// TwinCAT 3 PLC project PRG_B_Base_HMI
// Title: B_Base_HMI_Connector
// Company: RafalOS
// Author: Rafał Osajda
// ProjectVersion: 0.0.1.00
// ProgramVersion: 3.1.4026.18
// libraries:
//   B_Base, * (RafalOS)
//   Tc2_Standard, * (Beckhoff Automation GmbH)
//   Tc2_System, * (Beckhoff Automation GmbH)
//   Tc3_Module, * (Beckhoff Automation GmbH)
// project tree:
//   DUTs/ ST_BaseHMIDescriptor.TcDUT, ST_BaseHMIDescriptorEdit.TcDUT, ST_ListOfElement_HMI.TcDUT, ST_RowListOfElement_HMI.TcDUT
//   / PlcTask.TcTTO (not stored)
//   POUs Compilation/ PRG_Compilation.TcPOU
//   POUs/A02_FB_BaseHMILogger/ FB_BaseHMILogger.TcPOU, ITF_BaseHMILogger.TcIO, ST_BaseHMILogger.TcDUT
//   POUs/A03a_FB_BaseHMILoggerElement_View/ FB_BaseHMILoggerElement_View.TcPOU, ITF_BaseHMILoggerElement_View.TcIO, ST_BaseHMIConnectorEvents_ActionButtuns.TcDUT (not stored), ST_BaseHMIConnectorEvents_DetailInformation.TcDUT (not stored), ST_BaseHMIConnectorEvents_Filter.TcDUT (not stored), ST_BaseHMIConnectorEvents_ListToDisplay.TcDUT, ST_BaseHMILoggerElement_View.TcDUT, ST_BaseHMIConnectorEvents_ListToDisplayRow.TcDUT (not stored)
//   POUs/A03b_FB_BaseHMILoggerElement_Command/ FB_BaseHMILoggerElement_Command.TcPOU, ITF_BaseHMILoggerElement_Command.TcIO, ST_BaseHMILoggerElement_Command_DataCheck.TcDUT, ST_BaseHMILoggerElement_Command.TcDUT
//   POUs/A04a_FB_BaseHMIComponent_View/ FB_BaseHMIComponent_View.TcPOU, ITF_BaseHMIComponent_View.TcIO, ST_BaseHMIComponent_View.TcDUT, ST_BaseHMIComponent_View_Link.TcDUT
//   POUs/A04b_FB_BaseHMIComponent_Command/ FB_BaseHMIComponent_Command.TcPOU, ITF_BaseHMIComponent_Command.TcIO, ST_BaseHMIComponent_Command.TcDUT, ST_BaseHMIComponent_Command_Link.TcDUT
//   POUs/A05a_FB_BaseHMIControlElement_View/ FB_BaseHMIControlElement_View.TcPOU, ITF_BaseHMIControlElement_View.TcIO, ST_BaseHMIControlElement_View.TcDUT, ST_BaseHMIControlElement_View_Link.TcDUT
//   POUs/A05b_FB_BaseHMIControlElement_Command/ FB_BaseHMIControlElement_Command.TcPOU, ITF_BaseHMIControlElement_Command.TcIO, ST_BaseHMIControlElement_Command.TcDUT, ST_BaseHMIControlElement_Command_Link.TcDUT
//   POUs/A06a_FB_BaseHMIGroupElement_View/ FB_BaseHMIGroupElement_View.TcPOU, ITF_BaseHMIGroupElement_View.TcIO, ST_BaseHMIGroupElement_View.TcDUT, ST_BaseHMIGroupElement_View_Link.TcDUT
//   POUs/A06b_FB_BaseHMIGroupElement_Command/ FB_BaseHMIGroupElement_Command.TcPOU, ITF_BaseHMIGroupElement_Command.TcIO, ST_BaseHMIGroupElement_Command.TcDUT, ST_BaseHMIGroupElement_Command_Link.TcDUT
//   POUs/A07a_FB_BaseHMITopElement_View/ FB_BaseHMITopElement_View.TcPOU, ITF_BaseHMITopElement_View.TcIO, ST_BaseHMITopElement_View.TcDUT, ST_BaseHMITopElement_View_Link.TcDUT
//   POUs/A07b_FB_BaseHMITopElement_Command/ FB_BaseHMITopElement_Command.TcPOU, ITF_BaseHMITopElement_Command.TcIO, ST_BaseHMITopElement_Command.TcDUT, ST_BaseHMITopElement_Command_Link.TcDUT
//   POUs/B02_Recipe/ FB_BaseRecipe_HMI.TcPOU, ITF_BaseRecipe_HMI.TcIO, ST_BaseRecipe_HMI.TcDUT
// real-time tasks:
//   TASK PlcTask: cycle T#10ms, priority 20, ADS port 350

// ---- DUTs/ST_BaseHMIDescriptor.TcDUT
TYPE ST_BaseHMIDescriptor :
STRUCT
	wsText						: WSTRING;
	sUnit						: STRING(6);
	rValue						: REAL;
	rMin						: REAL;
	rMax						: REAL;
	rDefaultValue				: REAL;
END_STRUCT
END_TYPE

// ---- DUTs/ST_BaseHMIDescriptorEdit.TcDUT
TYPE ST_BaseHMIDescriptorEdit :
STRUCT
	wsText						: WSTRING;
	sUnit						: STRING(6);
	rValue						: REAL;
	rMin						: REAL;
	rMax						: REAL;
	rDefaultValue				: REAL;
	rValueOld					: REAL; //wartosc przed zmiana do porównania czy cos się zmieniło
	bSave						: BOOL;
	bSetDefault					: BOOL;
	bCancel						: BOOL;
	bVisibleSave				: BOOL;
	bVisibleSetDefault			: BOOL;
	bVisibleCancel				: BOOL;
	iID							: int; //numer deskryptora do edycji
END_STRUCT
END_TYPE

// ---- DUTs/ST_ListOfElement_HMI.TcDUT
TYPE ST_ListOfElement_HMI :
STRUCT
(*	Lista wszystkich dodanych komponentów 	*)
	arrRow					: ARRAY [1..GVL_BaseConstans.MAX_NUMBER_OF_ALL_ITEM] OF ST_RowListOfElement_HMI;
	iNumberOfAdded			: INT;
(*	Lista indeksów PB w tablicy arrWiersz	*)
	arrRowOfListTE			: ARRAY [1..GVL_BaseConstans.MAX_NUMBER_OF_TOP_ELEMENT] OF INT;
	iNumberOfAddedTE		: INT;
END_STRUCT
END_TYPE

// ---- DUTs/ST_RowListOfElement_HMI.TcDUT
TYPE ST_RowListOfElement_HMI :
STRUCT
	stIdentifiers		: ST_BaseElementIdentifier;
	itfElement			: ITF_BaseHMIComponent_View;
//
	arrChild			: ARRAY [0..GVL_BaseConstans.MAX_ITEM_PER_ELEMENT] OF INT;
	iNumberOfChildAdded	: INT;
	
END_STRUCT
END_TYPE

// ---- POUs/A02_FB_BaseHMILogger/ST_BaseHMILogger.TcDUT
TYPE ST_BaseHMILogger :
STRUCT
	bDanaBaseLogger		: BOOL;
END_STRUCT
END_TYPE

// ---- POUs/A03a_FB_BaseHMILoggerElement_View/ST_BaseHMIConnectorEvents_ListToDisplay.TcDUT
TYPE ST_BaseHMIConnectorEvents_ListToDisplay :
STRUCT
	arrToDisplay				: ARRAY [1..GVL_BaseConstans.MAX_EVENTS_TO_SHOW] OF ST_BaseHMIConnectorEvents_ListToDisplayRow;
	iNumberOfRow				: INT;

END_STRUCT
END_TYPE

// ---- POUs/A03a_FB_BaseHMILoggerElement_View/ST_BaseHMILoggerElement_View.TcDUT
TYPE ST_BaseHMILoggerElement_View :
STRUCT
	stFilter						: ST_BaseHMIConnectorEvents_Filter;
	stListOfEventsToDisplay			: ST_BaseHMIConnectorEvents_ListToDisplay;
	stButtons						: ST_BaseHMIConnectorEvents_ActionButtuns;
	stDetailInformation				: ST_BaseHMIConnectorEvents_DetailInformation;
	bSelected						: BOOL;
	iSelectedRow					: INT;
	iSelectedRowPrevius				: INT;
	bRefreshInfo					: BOOL;
	bRefreshList					: BOOL;
	
END_STRUCT
END_TYPE

// ---- POUs/A03b_FB_BaseHMILoggerElement_Command/ST_BaseHMILoggerElement_Command_DataCheck.TcDUT
TYPE ST_BaseHMILoggerElement_Command_DataCheck :
STRUCT
	eMode			: REFERENCE TO E_BaseMachineMode;	//tryb pracy
	bSafety			: REFERENCE TO BOOL;	//ogólna flaga czy safety pozwala na pracę 
END_STRUCT
END_TYPE

// ---- POUs/A03b_FB_BaseHMILoggerElement_Command/ST_BaseHMILoggerElement_Command.TcDUT
TYPE ST_BaseHMILoggerElement_Command :
STRUCT
END_STRUCT
END_TYPE

// ---- POUs/A04a_FB_BaseHMIComponent_View/ST_BaseHMIComponent_View.TcDUT
TYPE ST_BaseHMIComponent_View :
STRUCT
	wsName			: WSTRING;
	
END_STRUCT
END_TYPE

// ---- POUs/A04a_FB_BaseHMIComponent_View/ST_BaseHMIComponent_View_Link.TcDUT
(*			
	RAFALOS
	Rafał Osajda		23.09.2025		TC 4024.66
	Struktura pomocnicza potrzeba do wiazania zmiennych
*)
TYPE ST_BaseHMIComponent_View_Link :
STRUCT
	stLoggerElement				: ST_BaseHMILoggerElement_View;
	stComponent					: ST_BaseHMIComponent_View;
END_STRUCT
END_TYPE

// ---- POUs/A04b_FB_BaseHMIComponent_Command/ST_BaseHMIComponent_Command.TcDUT
TYPE ST_BaseHMIComponent_Command :
STRUCT
END_STRUCT
END_TYPE

// ---- POUs/A04b_FB_BaseHMIComponent_Command/ST_BaseHMIComponent_Command_Link.TcDUT
(*			
	RAFALOS
	Rafał Osajda		23.09.2025		TC 4024.66
	Struktura pomocnicza potrzeba do wiazania zmiennych
*)
TYPE ST_BaseHMIComponent_Command_Link :
STRUCT
	stLoggerElement				: ST_BaseHMILoggerElement_Command;
	stComponent					: ST_BaseHMIComponent_Command;
END_STRUCT
END_TYPE

// ---- POUs/A05a_FB_BaseHMIControlElement_View/ST_BaseHMIControlElement_View.TcDUT
TYPE ST_BaseHMIControlElement_View :
STRUCT
	bDanaBaseControlElement		: BOOL;
	
END_STRUCT
END_TYPE

// ---- POUs/A05a_FB_BaseHMIControlElement_View/ST_BaseHMIControlElement_View_Link.TcDUT
(*			
	RAFALOS
	Rafał Osajda		23.09.2025		TC 4024.66
	Struktura pomocnicza potrzeba do wiazania zmiennych
*)
TYPE ST_BaseHMIControlElement_View_Link :
STRUCT
	stLoggerElement				: ST_BaseHMILoggerElement_View;
	stComponent					: ST_BaseHMIComponent_View;
	stControlElement			: ST_BaseHMIControlElement_View;
END_STRUCT
END_TYPE

// ---- POUs/A05b_FB_BaseHMIControlElement_Command/ST_BaseHMIControlElement_Command.TcDUT
TYPE ST_BaseHMIControlElement_Command :
STRUCT
END_STRUCT
END_TYPE

// ---- POUs/A05b_FB_BaseHMIControlElement_Command/ST_BaseHMIControlElement_Command_Link.TcDUT
TYPE ST_BaseHMIControlElement_Command_Link :
STRUCT
	stLoggerElement				: ST_BaseHMILoggerElement_Command;
	stComponent					: ST_BaseHMIComponent_Command;
	stControlElement			: ST_BaseHMIControlElement_Command;
END_STRUCT
END_TYPE

// ---- POUs/A06a_FB_BaseHMIGroupElement_View/ST_BaseHMIGroupElement_View.TcDUT
TYPE ST_BaseHMIGroupElement_View :
STRUCT
	bDanaBaseGroupElement		: BOOL;
END_STRUCT
END_TYPE

// ---- POUs/A06a_FB_BaseHMIGroupElement_View/ST_BaseHMIGroupElement_View_Link.TcDUT
(*			
	RAFALOS
	Rafał Osajda		23.09.2025		TC 4024.66
	Struktura pomocnicza potrzeba do wiazania zmiennych
*)
TYPE ST_BaseHMIGroupElement_View_Link :
STRUCT
	stLoggerElement				: ST_BaseHMILoggerElement_View;
	stComponent					: ST_BaseHMIComponent_View;
	stControlElement			: ST_BaseHMIControlElement_View;
	stGroupElement				: ST_BaseHMIGroupElement_View;
END_STRUCT
END_TYPE

// ---- POUs/A06b_FB_BaseHMIGroupElement_Command/ST_BaseHMIGroupElement_Command.TcDUT
TYPE ST_BaseHMIGroupElement_Command :
STRUCT
END_STRUCT
END_TYPE

// ---- POUs/A06b_FB_BaseHMIGroupElement_Command/ST_BaseHMIGroupElement_Command_Link.TcDUT
TYPE ST_BaseHMIGroupElement_Command_Link :
STRUCT
	stLoggerElement				: ST_BaseHMILoggerElement_Command;
	stComponent					: ST_BaseHMIComponent_Command;
	stControlElement			: ST_BaseHMIControlElement_Command;
	stGroupElement				: ST_BaseHMIGroupElement_Command;
END_STRUCT
END_TYPE

// ---- POUs/A07a_FB_BaseHMITopElement_View/ST_BaseHMITopElement_View.TcDUT
TYPE ST_BaseHMITopElement_View :
STRUCT
	bDanaTopElement				: BOOL;
END_STRUCT
END_TYPE

// ---- POUs/A07a_FB_BaseHMITopElement_View/ST_BaseHMITopElement_View_Link.TcDUT
(*			
	RAFALOS
	Rafał Osajda		23.09.2025		TC 4024.66
	Struktura pomocnicza potrzeba do wiazania zmiennych
*)
TYPE ST_BaseHMITopElement_View_Link :
STRUCT
	stLoggerElement				: ST_BaseHMILoggerElement_View;
	stComponent					: ST_BaseHMIComponent_View;
	stControlElement			: ST_BaseHMIControlElement_View;
	stGroupElement				: ST_BaseHMIGroupElement_View;
	stTopElement				: ST_BaseHMITopElement_View;
END_STRUCT
END_TYPE

// ---- POUs/A07b_FB_BaseHMITopElement_Command/ST_BaseHMITopElement_Command.TcDUT
TYPE ST_BaseHMITopElement_Command :
STRUCT
END_STRUCT
END_TYPE

// ---- POUs/A07b_FB_BaseHMITopElement_Command/ST_BaseHMITopElement_Command_Link.TcDUT
TYPE ST_BaseHMITopElement_Command_Link :
STRUCT
	stLoggerElement				: ST_BaseHMILoggerElement_Command;
	stComponent					: ST_BaseHMIComponent_Command;
	stControlElement				: ST_BaseHMIControlElement_Command;
	stGroupElement				: ST_BaseHMIGroupElement_Command;
	stTopElement					: ST_BaseHMITopElement_Command;
END_STRUCT
END_TYPE

// ---- POUs/B02_Recipe/ST_BaseRecipe_HMI.TcDUT
TYPE ST_BaseRecipe_HMI :
STRUCT
END_STRUCT
END_TYPE

// ---- POUs/A02_FB_BaseHMILogger/ITF_BaseHMILogger.TcIO
INTERFACE ITF_BaseHMILogger

END_INTERFACE

// ---- POUs/A03a_FB_BaseHMILoggerElement_View/ITF_BaseHMILoggerElement_View.TcIO
INTERFACE ITF_BaseHMILoggerElement_View

(*			
	RafalOS
	Rafał Osajda		19.11.2025		TC 4024.66
	Czyści danych przy zmienia ramki po poprzedniej ramce
*)
METHOD PUBLIC ClearAfterScreen : BOOL
VAR_INPUT
END_VAR
END_METHOD

(*			
	EVERDE sp. z o.o.
	Rafał Osajda		09.09.2025		TC 4024.66
	Generuje tablicę zdarzeń dla podanego ID dla 0 dla wszystkich elementów
*)
METHOD PUBLIC GetEventTableForIDItem : BOOL
VAR_INPUT
	uiIdItem			: UINT;
END_VAR
END_METHOD

(*			
	EVERDE sp. z o.o.
	Rafał Osajda		09.09.2025		TC 4024.66
	Zwraca tablicę swoich zdarzeń
*)
METHOD PUBLIC GetYourEventTable : BOOL
VAR_INPUT
END_VAR
END_METHOD

(*			
	RafalOS
	Rafał Osajda		14.11.2025		TC 4024.66
	Metoda przygotowywania danych dla HMI 
	W niej odbywa się odpytywanie właściego elementu przez łącznik
*)
METHOD PUBLIC PrepareDataForHMI : BOOL
VAR_INPUT
END_VAR
END_METHOD

(*			
	RafalOS
	Rafał Osajda		19.11.2025		TC 4024.66
	Przygotowanie ramki pood tamke do wyświetlenia - tylko przygotowanie a nie przygotowanie danych do wyświetlenia
*)
METHOD PUBLIC PrepareForScreen : BOOL
VAR_INPUT
END_VAR
END_METHOD

END_INTERFACE

// ---- POUs/A03b_FB_BaseHMILoggerElement_Command/ITF_BaseHMILoggerElement_Command.TcIO
INTERFACE ITF_BaseHMILoggerElement_Command

END_INTERFACE

// ---- POUs/A04a_FB_BaseHMIComponent_View/ITF_BaseHMIComponent_View.TcIO
INTERFACE ITF_BaseHMIComponent_View EXTENDS ITF_BaseHMILoggerElement_View

METHOD PUBLIC IsValidCommonData : BOOL
VAR_INPUT
END_VAR
END_METHOD

METHOD PUBLIC JoinTheList : INT
VAR_INPUT
	refstList				: REFERENCE TO ST_ListOfElement_HMI;
	iNumberOfParent			: INT; 	//numer rodzica na liście
END_VAR
END_METHOD

METHOD PUBLIC LinkCommonData : BOOL
VAR_INPUT
	stCommonData				: REFERENCE TO ST_BaseCommonData;
END_VAR
END_METHOD

END_INTERFACE

// ---- POUs/A04b_FB_BaseHMIComponent_Command/ITF_BaseHMIComponent_Command.TcIO
INTERFACE ITF_BaseHMIComponent_Command EXTENDS ITF_BaseHMILoggerElement_Command

END_INTERFACE

// ---- POUs/A05a_FB_BaseHMIControlElement_View/ITF_BaseHMIControlElement_View.TcIO
INTERFACE ITF_BaseHMIControlElement_View EXTENDS ITF_BaseHMIComponent_View

END_INTERFACE

// ---- POUs/A05b_FB_BaseHMIControlElement_Command/ITF_BaseHMIControlElement_Command.TcIO
INTERFACE ITF_BaseHMIControlElement_Command EXTENDS ITF_BaseHMIComponent_Command

END_INTERFACE

// ---- POUs/A06a_FB_BaseHMIGroupElement_View/ITF_BaseHMIGroupElement_View.TcIO
INTERFACE ITF_BaseHMIGroupElement_View EXTENDS ITF_BaseHMIControlElement_View

END_INTERFACE

// ---- POUs/A06b_FB_BaseHMIGroupElement_Command/ITF_BaseHMIGroupElement_Command.TcIO
INTERFACE ITF_BaseHMIGroupElement_Command EXTENDS ITF_BaseHMIControlElement_Command

END_INTERFACE

// ---- POUs/A07a_FB_BaseHMITopElement_View/ITF_BaseHMITopElement_View.TcIO
INTERFACE ITF_BaseHMITopElement_View EXTENDS ITF_BaseHMIComponent_View

END_INTERFACE

// ---- POUs/A07b_FB_BaseHMITopElement_Command/ITF_BaseHMITopElement_Command.TcIO
INTERFACE ITF_BaseHMITopElement_Command EXTENDS ITF_BaseHMIGroupElement_Command

END_INTERFACE

// ---- POUs/B02_Recipe/ITF_BaseRecipe_HMI.TcIO
INTERFACE ITF_BaseRecipe_HMI EXTENDS ITF_Base

(*			
	RafalOS
	Rafał Osajda		03.03.2025		TC 4026.13		wer. 0.0.0.1
	Kopiuje składniki z wybranej receptury i tworzy nową recepture
*)
METHOD PUBLIC AddRecipeFromRecipe : BOOL
VAR_INPUT
	uiNumberRecipe				: UINT;
	stTexts						: ST_BaseLabel;
END_VAR
END_METHOD

(*			
	RafalOS
	Rafał Osajda		03.03.2025		TC 4026.13		wer. 0.0.0.1
	Kopiuje składniki z wybranego szablonu i tworzy nową recepture
*)
METHOD PUBLIC AddRecipeFromTemplate : BOOL
VAR_INPUT
	uiNumberTemplates			: UINT;
	stTexts						: ST_BaseLabel;
END_VAR
END_METHOD

(*			
	RafalOS
	Rafał Osajda		03.06.2025		TC 4024.66
	usuwa referencje do wybranej
*)
METHOD PUBLIC ClearChosen
VAR_INPUT
END_VAR
END_METHOD

(*			
	RafalOS
	Rafał Osajda		25.10.2025		TC 4024.66
	Utworzenie nowych szablonów receptur na podstawie dodanych fb zewnętrznych - wywołanie metody powoduje
	skosowanie dotychczasowych szablonów i receptur
*)
METHOD PUBLIC CreateRecipeTemplates : BOOL
VAR_INPUT
END_VAR
END_METHOD

(*			
	RafalOS
	Rafał Osajda		03.03.2025		TC 4026.13		wer. 0.0.0.1
	
*)
METHOD PUBLIC DeleteRecipe : BOOL
VAR_INPUT
	uiNumber				: uint;
END_VAR
END_METHOD

(*			
	RafalOS
	Rafał Osajda		03.03.2025		TC 4026.13		wer. 0.0.0.1
	
*)
METHOD PUBLIC GetIngredientFromRecipe : ST_BaseDescriptor
VAR_INPUT
	uiNumberOfRecipe			: UINT;
	uiNumberOfIngredient		: UINT;
END_VAR
END_METHOD

(*			
	RafalOS
	Rafał Osajda		02.12.2025		TC 4024.66
	Zwraca do tablicy wybrany zakres składników
*)
METHOD PUBLIC GetIngredientRange 
VAR_INPUT
	iRecipe			: INT;	//numer receptury z której bierzemy składniki
	iStartIndex		: INT;	//numer startowy składnika
	iCount			: INT;	//ilośc pobieranych 
END_VAR
VAR_IN_OUT
	arrOut : ARRAY [*] OF ST_BaseDescriptor;
END_VAR
VAR_OUTPUT
	iNumberOfFilledData	: INT;	//ilosc wypelnionych danych na strone
END_VAR
END_METHOD

METHOD GetNameList : ST_BaseRecipeList
VAR_INPUT
END_VAR
END_METHOD

METHOD GetNameListTemplate : ST_BaseRecipeList
VAR_INPUT
END_VAR
END_METHOD

METHOD GetNamesOfSelectRecipe : ST_BaseLabel
VAR_INPUT

END_VAR
END_METHOD

(*			
	RafalOS
	Rafał Osajda		03.03.2025		TC 4026.13		wer. 0.0.0.1
	
*)
METHOD PUBLIC GetNumberIngredientOfRecipe : UINT
VAR_INPUT
	uiNumber				: UINT;
END_VAR
END_METHOD

METHOD PUBLIC GetNumberOfChoosen : UINT
VAR_INPUT
END_VAR
END_METHOD

METHOD PUBLIC GetNumberOfRecipe : UINT
VAR_INPUT
END_VAR
END_METHOD

METHOD PUBLIC GetNumberOfTemplate : UINT
VAR_INPUT
END_VAR
END_METHOD

(*			
	RafalOS
	Rafał Osajda		06.12.2025		TC 4024.66
	Sprawdza czy receptrua została wybrana
*)
METHOD PUBLIC IsRecipeSelected : BOOL
VAR_INPUT
END_VAR
END_METHOD

METHOD PUBLIC LinkRecipeDataHMI : BOOL
VAR_INPUT
	stRecipe			: REFERENCE TO ST_BaseRecipe_HMI;
END_VAR
END_METHOD

(*			
	RafalOS
	Rafał Osajda		06.12.2025		TC 4024.66
	Wybranie receputury
*)
METHOD SelectRecipe : BOOL
VAR_INPUT
	uiRecipe: UINT;
END_VAR
END_METHOD

(*			
	RafalOS
	Rafał Osajda		05.12.2025		TC 4024.66
	Ustawia nową wartośc w podanym składniku
*)
METHOD PUBLIC SetIngredientValue
VAR_INPUT
	iRecipe			: int;
	iIngredient		: INT;
	rValue			: REAL;
END_VAR
END_METHOD

END_INTERFACE

// ---- POUs Compilation/PRG_Compilation.TcPOU
PROGRAM PRG_Compilation
VAR
	fbLoggerHMI				: FB_BaseHMILogger;
	fbLoggerElementHMIView	: FB_BaseHMILoggerElement_View;
	fbLoggerElementHMICmd	: FB_BaseHMILoggerElement_Command;
	fbComponentHMIView		: FB_BaseHMIComponent_View;
	fbComponentHMICmd		: FB_BaseHMIComponent_Command;
	fbControlElementHMIView	: FB_BaseHMIControlElement_View;
	fbControlElementHMICmd	: FB_BaseHMIControlElement_Command;
	fbGroupElementHMIView	: FB_BaseHMIGroupElement_View;
	fbGroupElementHMICmd	: FB_BaseHMIGroupElement_Command;
	fbTopElementHMIView		: FB_BaseHMITopElement_View;
	fbTopElementHMICmd		: FB_BaseHMITopElement_Command;
	
	fbRecipe				: FB_BaseRecipe;
	fbRecipeHMI				: FB_BaseRecipe_HMI (fbBaseRecipe := fbRecipe);
END_VAR

END_PROGRAM

// ---- POUs/A02_FB_BaseHMILogger/FB_BaseHMILogger.TcPOU
(* póki co ten FB jest zbędny ale zostawiam jakby co*)
FUNCTION_BLOCK FB_BaseHMILogger// EXTENDS FB_Base IMPLEMENTS ITF_BaseLoggerElement_HMI
VAR
//	itfBaseLoggerConnector			: ITF_BaseLogger_HMI_Connector;	//łącznik bezpośredni do Logera
//	refstBaseLoggerDataHMI			: REFERENCE TO ST_BaseLogger_HMI;
END_VAR

END_FUNCTION_BLOCK

// ---- POUs/A03a_FB_BaseHMILoggerElement_View/FB_BaseHMILoggerElement_View.TcPOU
FUNCTION_BLOCK FB_BaseHMILoggerElement_View EXTENDS FB_Base IMPLEMENTS ITF_BaseHMILoggerElement_View
VAR
	itfBaseLoggerConnector					: ITF_BaseLogger_HMI_Connector_View;	//bezpośredni łącznik do logera odczyt danych
	itfBaseLoggerElementConnector			: ITF_BaseLoggerElement_HMI_Connector_View;	//lacznik do FB_BaseLoggerElement np zeby wyciągnąć identyfikator odczyt danych
	refstBaseLoggerElementDataHMI			: REFERENCE TO ST_BaseHMILoggerElement_View;
	refstMemoryEvents						: REFERENCE TO ST_BaseEvents_Memory;	//referencja do tablicy zgłoszeń
	bIsInit									: BOOL;	//flaga informująca czy wszystkie interfejsy są dobrze przypisane
	bIsValidData							: bool;	//flaga informująca czy wszystkie dane sa podpięte 
END_VAR

(*			
	RafalOS
	Rafał Osajda		19.11.2025		TC 4024.66
	Czyści danych przy zmienia ramki po poprzedniej ramce
*)
METHOD PUBLIC ClearAfterScreen : BOOL
VAR_INPUT
END_VAR
END_METHOD

METHOD PRIVATE CompleteTheDetailedInformation : BOOL
VAR_INPUT
	stRow			: ST_BaseHMIConnectorEvents_ListToDisplayRow;
END_VAR
THIS^.refstBaseLoggerElementDataHMI.stDetailInformation.uiIDEvent						:= stRow.uiIDEvent;
THIS^.refstBaseLoggerElementDataHMI.stDetailInformation.uiIDItem						:= stRow.uiIDItem;
THIS^.refstBaseLoggerElementDataHMI.stDetailInformation.sCode							:= stRow.sCode;
THIS^.refstBaseLoggerElementDataHMI.stDetailInformation.bActive							:= stRow.bActive;
THIS^.refstBaseLoggerElementDataHMI.stDetailInformation.bIgnoreRepetitions				:= stRow.bIgnoreRepetitions;
THIS^.refstBaseLoggerElementDataHMI.stDetailInformation.uiRepetitionCounter				:= stRow.uiRepetitionCounter;
THIS^.refstBaseLoggerElementDataHMI.stDetailInformation.sStart							:= stRow.sStart;
THIS^.refstBaseLoggerElementDataHMI.stDetailInformation.sFinish							:= stRow.sFinish;
THIS^.refstBaseLoggerElementDataHMI.stDetailInformation.sConfirmed						:= stRow.sConfirmed;
THIS^.refstBaseLoggerElementDataHMI.stDetailInformation.bConfirm						:= stRow.bConfirm;
THIS^.refstBaseLoggerElementDataHMI.stDetailInformation.bConfirmed						:= stRow.bConfirmed;
THIS^.refstBaseLoggerElementDataHMI.stDetailInformation.sEventCategory					:= stRow.sEventCategory;
THIS^.refstBaseLoggerElementDataHMI.stDetailInformation.wsDescription					:= stRow.wsDescription;
THIS^.refstBaseLoggerElementDataHMI.stDetailInformation.wsDescriptionFull				:= stRow.wsDescriptionFull;
END_METHOD

METHOD PRIVATE CopyDataToDisplay : BOOL
VAR_INPUT
	refarrToDisplay				: REFERENCE TO ARRAY [1..GVL_BaseConstans.MAX_EVENTS_TO_SHOW] OF ST_BaseHMIConnectorEvents_ListToDisplayRow;
	iNumberOfRow				: INT;
	stRowFromMemory				: ST_BaseEvents_RowInMemory;
	stItemInformation			: ST_BaseLogger_ItemDataToDisplay;
END_VAR
VAR
	wstmpDescriptionFull		: WSTRING;
	wstmpDescription			: WSTRING;
	iDltmp						: INT;
END_VAR
refarrToDisplay [iNumberOfRow].uiIDEvent			:= stRowFromMemory.uiIDEvent;
refarrToDisplay [iNumberOfRow].uiIDItem				:= stRowFromMemory.uiIDItem;
refarrToDisplay [iNumberOfRow].bActive				:= stRowFromMemory.bActive;
refarrToDisplay [iNumberOfRow].sCode				:= stItemInformation.sCode; 
refarrToDisplay [iNumberOfRow].bIgnoreRepetitions	:= stRowFromMemory.bIgnoreRepetitions;
refarrToDisplay [iNumberOfRow].bConfirm				:= stRowFromMemory.bConfirm;
refarrToDisplay [iNumberOfRow].bConfirmed			:= stRowFromMemory.bConfirmed;

refarrToDisplay [iNumberOfRow].sStart				:= THIS^.refstCommonData.itfTime.BaseDTToString (inDT := stRowFromMemory.dtStart);
IF (TO_STRING (stRowFromMemory.dtConfirmed) <> 'DT#1970-01-01-00:00:00') THEN
	refarrToDisplay [iNumberOfRow].sConfirmed		:= THIS^.refstCommonData.itfTime.BaseDTToString (inDT := stRowFromMemory.dtConfirmed);
ELSE
	refarrToDisplay [iNumberOfRow].sConfirmed		:= '';
END_IF
IF (TO_STRING (TO_STRING (stRowFromMemory.dtFinish)) <> 'DT#1970-01-01-00:00:00') THEN
	refarrToDisplay [iNumberOfRow].sFinish			:= THIS^.refstCommonData.itfTime.BaseDTToString (inDT := stRowFromMemory.dtFinish);
ELSE
	refarrToDisplay [iNumberOfRow].sFinish			:= '';
END_IF

refarrToDisplay [iNumberOfRow].sEventCategory		:= stItemInformation.sEventCategory; 
refarrToDisplay [iNumberOfRow].uiRepetitionCounter	:= stItemInformation.uiRepetitionCounter;
wstmpDescriptionFull		:= THIS^.GetTextFromLabelForActiveLocation (stLabel	:= stItemInformation.stDescription);
iDltmp												:= WLEN (wstmpDescriptionFull);
IF (iDltmp > 100) THEN
	wstmpDescription								:= WDELETE (wstmpDescriptionFull, iDltmp - 100, iDltmp);
END_IF
refarrToDisplay [iNumberOfRow].wsDescription		:= wstmpDescription;
refarrToDisplay [iNumberOfRow].wsDescriptionFull	:= wstmpDescriptionFull;
refarrToDisplay [iNumberOfRow].wsNameOfitem			:= THIS^.GetTextFromLabelForActiveLocation (stLabel := stItemInformation.stItemName);
END_METHOD

METHOD PUBLIC CreateLinkToEventsMemory : BOOL
VAR_INPUT
END_VAR
THIS^.refstMemoryEvents	REF= THIS^.itfBaseLoggerConnector.GetReferenceToStmemory ();


IF (__ISVALIDREF (THIS^.refstMemoryEvents)) THEN
	CreateLinkToEventsMemory		:= TRUE;
ELSE
	CreateLinkToEventsMemory		:= FALSE;
END_IF
END_METHOD

(*			
	EVERDE sp. z o.o.
	Rafał Osajda		09.09.2025		TC 4024.66
	Generuje tablicę zdarzeń dla podanego ID dla 0 dla wszystkich elementów
*)
METHOD PUBLIC GetEventTableForIDItem : BOOL
VAR_INPUT
	uiIdItem				: UINT;
END_VAR
VAR_INST
	bFilterIsActivePrevius	: BOOL;	
END_VAR
VAR
	iI						: INT;
	bFilterIsActive			: BOOL;
	bUsunZListy				: BOOL;
	btmpUsunZListy			: BOOL;
	refstMemory				: REFERENCE TO ST_BaseEvents_Memory;
	refstListToDisplay		: REFERENCE TO ST_BaseHMIConnectorEvents_ListToDisplay;
	refstFilter				: REFERENCE TO ST_BaseHMIConnectorEvents_Filter;
	refstActionButtons		: REFERENCE TO ST_BaseHMIConnectorEvents_ActionButtuns;
	stRowFromMemory			: ST_BaseEvents_RowInMemory;
	stItemInformation		: ST_BaseLogger_ItemDataToDisplay;
(*	Ilosci zdarzen wyswietlanych na liscie	*)
	stNumberEventToDisplay	: ST_BaseEvents_ActiveEvents;
//
	iIAck: INT;
	iIClose: INT;
END_VAR
(*
	sprawdzenie czy jest coś nowego - tak generuj
	jak już jest wygenerowana jakaś lista i zmienił się filtr - tak to generuj

*)
IF (THIS^.refstMemoryEvents.iNumberOfRow > 0) THEN

	refstMemory				REF= THIS^.refstMemoryEvents;
	refstListToDisplay		REF= THIS^.refstBaseLoggerElementDataHMI.stListOfEventsToDisplay;
	refstFilter				REF= THIS^.refstBaseLoggerElementDataHMI.stFilter;
	refstActionButtons		REF= THIS^.refstBaseLoggerElementDataHMI.stButtons;
	bFilterIsActive			:= GetIsActiveFilter (refstFilter := refstFilter);		//sprawdzenie czy jest aktywny filtr
	
	IF (THIS^.itfBaseLoggerConnector.GetChangeInMemory () OR bFilterIsActive 
		OR bFilterIsActivePrevius OR THIS^.refstBaseLoggerElementDataHMI.bRefreshList) THEN
		THIS^.refstBaseLoggerElementDataHMI.bRefreshList	:= FALSE;
		bFilterIsActivePrevius								:= bFilterIsActive;

		THIS^.itfBaseLoggerConnector.ResetChangeInMemory ();
		(*	Wyczyszczenie tablicy wyświetlania		*)
		Tc2_System.MEMSET (
			destAddr		:= ADR (refstListToDisplay.arrToDisplay),
			fillByte		:= 0,
			n				:= SIZEOF (refstListToDisplay.arrToDisplay)
		);
		refstListToDisplay.iNumberOfRow		:= 0;
		FOR iI := 1 TO refstMemory.iNumberOfRow DO
			IF (uiIdItem = refstMemory.arrRow [iI].uiIDItem OR uiIdItem = 0) THEN
				stRowFromMemory			:= refstMemory.arrRow [iI];
				stItemInformation		:= THIS^.itfBaseLoggerConnector.GetInformationFromItem (uiIDItem := uiIdItem, uiIDEvent := stRowFromMemory.uiIDEvent);
				bUsunZListy		:= THIS^.RemoveRowFormList (
										refstFilter 		:= refstFilter, 
										uiIDEvent 			:= stRowFromMemory.uiIDEvent, 
										uiIDItem 			:=  stRowFromMemory.uiIDItem,
										bActive				:= stRowFromMemory.bActive,
										stItemInformation	:= stItemInformation
									);
				IF (NOT bUsunZListy) THEN
					refstListToDisplay.iNumberOfRow		:= refstListToDisplay.iNumberOfRow + 1;
					THIS^.CopyDataToDisplay (
						refarrToDisplay					:= refstListToDisplay.arrToDisplay,
						iNumberOfRow					:= refstListToDisplay.iNumberOfRow,
						stRowFromMemory					:= stRowFromMemory,
						stItemInformation				:= stItemInformation
					);
	(*	Informacja o ilosciach zgloszen na wyswietlanej liście 		*)
					stNumberEventToDisplay.iTotalNumer	:= stNumberEventToDisplay.iTotalNumer + 1;
					IF (refstListToDisplay.arrToDisplay [refstListToDisplay.iNumberOfRow].bActive) THEN
						stNumberEventToDisplay.iNumberOfActive	:= stNumberEventToDisplay.iNumberOfActive + 1;
						stNumberEventToDisplay.arrNumberOfActive [stItemInformation.eEventCategory] := stNumberEventToDisplay.arrNumberOfActive [stItemInformation.eEventCategory] + 1;
						stNumberEventToDisplay.arrActive [stItemInformation.eEventCategory]	:= TRUE;
					END_IF
					IF (refstListToDisplay.arrToDisplay [refstListToDisplay.iNumberOfRow].bConfirm AND 
						NOT refstListToDisplay.arrToDisplay [refstListToDisplay.iNumberOfRow].bConfirmed) THEN
						stNumberEventToDisplay.iNumberOfActiveWithConfirmation	:= stNumberEventToDisplay.iNumberOfActiveWithConfirmation + 1;
					END_IF
					stNumberEventToDisplay.arrTotalNumer [stItemInformation.eEventCategory] := stNumberEventToDisplay.arrTotalNumer [stItemInformation.eEventCategory] + 1;
				END_IF	//usuwanie z listy
			END_IF
	(*	Liczba zgłoszeń większa od tych co wyświetlamy	starsze można zobaczyć na kompie po podłaczeniu 	*)
			IF (refstListToDisplay.iNumberOfRow = TO_INT (GVL_BaseConstans.MAX_EVENTS_TO_SHOW)) THEN
				EXIT;
			END_IF
		END_FOR	//koniec przechodzenia przez wiersze pamięci
	(*	Informacja o ilosciach zgloszen		*)
		IF (uiIdItem > 0) THEN
			THIS^.PrepareQuantitiesForDisplay (
				stCounted		:= stNumberEventToDisplay,
				stFromLogger	:= THIS^.itfBaseLoggerConnector.GetEventCountsForItem (uiIDItem := uiIDItem)
			);
		ELSE
			THIS^.PrepareQuantitiesForDisplay (
				stCounted		:= stNumberEventToDisplay,
				stFromLogger	:= THIS^.itfBaseLoggerConnector.GetEventCounts ()
			);
		END_IF
		refstActionButtons.bAcknowledgeAllActive	:= stNumberEventToDisplay.iNumberOfActiveWithConfirmation > 0;
		refstActionButtons.bCloseAllActive			:= stNumberEventToDisplay.iNumberOfActive > 0;
	END_IF
	IF (THIS^.refstBaseLoggerElementDataHMI.bSelected) THEN
		refstActionButtons.bAcknowledgeSelectedActive	:= refstListToDisplay.arrToDisplay [THIS^.refstBaseLoggerElementDataHMI.iSelectedRow].bConfirm AND 
			NOT refstListToDisplay.arrToDisplay [THIS^.refstBaseLoggerElementDataHMI.iSelectedRow].bConfirmed;
		refstActionButtons.bCloseSelectedActive			:= refstListToDisplay.arrToDisplay [THIS^.refstBaseLoggerElementDataHMI.iSelectedRow].bConfirm AND 
			refstListToDisplay.arrToDisplay [THIS^.refstBaseLoggerElementDataHMI.iSelectedRow].bConfirmed;
	ELSE
		refstActionButtons.bAcknowledgeSelectedActive	:= FALSE;
		refstActionButtons.bCloseSelectedActive			:= FALSE;
	END_IF
	
	(*	Wybor zgloszenia z listy	*)

	IF ((THIS^.refstBaseLoggerElementDataHMI.iSelectedRow <> THIS^.refstBaseLoggerElementDataHMI.iSelectedRowPrevius AND
		THIS^.refstBaseLoggerElementDataHMI.bSelected) OR THIS^.refstBaseLoggerElementDataHMI.bRefreshInfo ) THEN
		THIS^.CompleteTheDetailedInformation (stRow := refstListToDisplay.arrToDisplay [THIS^.refstBaseLoggerElementDataHMI.iSelectedRow]);
	ELSIF (NOT THIS^.refstBaseLoggerElementDataHMI.bSelected) THEN
		THIS^.refstBaseLoggerElementDataHMI.iSelectedRow		:= -1;
		THIS^.refstBaseLoggerElementDataHMI.iSelectedRowPrevius	:= -1;
	END_IF 
	
	(*	Obsługa przycisków zamykania i potwierrdzania zgłoszeń	*)

	IF (THIS^.refstBaseLoggerElementDataHMI.stButtons.bAcknowledgeSelected) THEN //potwierdz zgłoszenie
		IF (refstListToDisplay.arrToDisplay [THIS^.refstBaseLoggerElementDataHMI.iSelectedRow].bConfirm AND 
			NOT refstListToDisplay.arrToDisplay [THIS^.refstBaseLoggerElementDataHMI.iSelectedRow].bConfirmed) THEN
			THIS^.itfBaseLoggerElementConnector.EventAcknowledgeByID (uiIDEvent := THIS^.refstBaseLoggerElementDataHMI.stDetailInformation.uiIDEvent);
		END_IF
	END_IF

	IF (THIS^.refstBaseLoggerElementDataHMI.stButtons.bCloseSelected) THEN	//zamknij zgłoszenie
		IF (refstListToDisplay.arrToDisplay [THIS^.refstBaseLoggerElementDataHMI.iSelectedRow].bActive OR 
			refstListToDisplay.arrToDisplay [THIS^.refstBaseLoggerElementDataHMI.iSelectedRow].sFinish <> '') THEN
			THIS^.itfBaseLoggerElementConnector.EventSetInactiveByID (uiIDEvent := THIS^.refstBaseLoggerElementDataHMI.stDetailInformation.uiIDEvent);
		END_IF
	END_IF

	IF (THIS^.refstBaseLoggerElementDataHMI.stButtons.bAcknowledgeAll) THEN //potwierdz wszystkie niepotwierdzone zgłoszenie
		FOR iIAck := 1 TO TO_INT (refstListToDisplay.iNumberOfRow) DO
			IF (refstListToDisplay.arrToDisplay [iIAck].bConfirm AND 
				NOT refstListToDisplay.arrToDisplay [iIAck].bConfirmed) THEN
				THIS^.itfBaseLoggerElementConnector.EventAcknowledgeByID (uiIDEvent := refstListToDisplay.arrToDisplay [iIAck].uiIDEvent);
			END_IF
		END_FOR
	END_IF
	IF (THIS^.refstBaseLoggerElementDataHMI.stButtons.bCloseAll) THEN	//zamknij wszystkie nie zamnknięte zgłoszenie
		FOR iIClose := 1 TO TO_INT (refstListToDisplay.iNumberOfRow) DO
			IF (refstListToDisplay.arrToDisplay [iIClose].bActive OR refstListToDisplay.arrToDisplay [iIClose].sFinish <> '') THEN
				THIS^.itfBaseLoggerElementConnector.EventSetInactiveByID (uiIDEvent := refstListToDisplay.arrToDisplay [iIClose].uiIDEvent);
			END_IF
		END_FOR
	END_IF
	
	
	THIS^.refstBaseLoggerElementDataHMI.bRefreshList		:= 	refstActionButtons.bAcknowledgeSelected OR
																refstActionButtons.bCloseSelected OR
																refstActionButtons.bAcknowledgeAll OR
																refstActionButtons.bCloseAll;
	THIS^.refstBaseLoggerElementDataHMI.bRefreshInfo		:= 	refstActionButtons.bAcknowledgeSelected	OR
																refstActionButtons.bCloseSelected OR
	                                                          	refstActionButtons.bAcknowledgeAll OR
                                                               	refstActionButtons.bCloseAll;
	refstActionButtons.bAcknowledgeSelected					:= FALSE;
	refstActionButtons.bCloseSelected						:= FALSE;
	refstActionButtons.bAcknowledgeAll						:= FALSE;
	refstActionButtons.bCloseAll							:= FALSE;

END_IF
END_METHOD

METHOD PRIVATE GetIsActiveFilter : BOOL
VAR_INPUT
	refstFilter				: REFERENCE TO ST_BaseHMIConnectorEvents_Filter;
END_VAR
VAR
	bResult: BOOL;
	iI: INT;
END_VAR
bResult				:= refstFilter.bActive OR 
						refstFilter.bNotActive OR
						refstFilter.bIDEvent OR
						refstFilter.bIDItem;
FOR iI := 1 TO GVL_BaseConstans.NUMBER_OF_EVENT_CATEGORIES DO
	bResult			:= bResult OR refstFilter.arrSelectedEventCategory [iI];
END_FOR

GetIsActiveFilter	:= bResult;
END_METHOD

METHOD PROTECTED GetTextFromLabel : WSTRING
VAR_INPUT
	stLabel				: ST_BaseLabel;
	eLocation			: E_BaseLocation;
END_VAR
GetTextFromLabel := stLabel.arrText [eLocation];
END_METHOD

METHOD PROTECTED GetTextFromLabelForActiveLocation : WSTRING
VAR_INPUT
	stLabel				: ST_BaseLabel;
END_VAR

VAR
	dfsfsdaf: WSTRING;
END_VAR
GetTextFromLabelForActiveLocation := stLabel.arrText [THIS^.refstCommonData.itfLocaciotn.GetLocation ()];
END_METHOD

(*			
	EVERDE sp. z o.o.
	Rafał Osajda		09.09.2025		TC 4024.66
	Zwraca tablicę swoich zdarzeń
*)
METHOD PUBLIC GetYourEventTable : BOOL
VAR_INPUT
END_VAR
THIS^.GetEventTableForIDItem (uiIdItem := THIS^.itfBaseLoggerElementConnector.GetID ());		//przygotowanie tablicy dla siebie
END_METHOD

(*			
	RAFALOS
	Rafał Osajda		23.09.2025		TC 4024.66
	Zwraca informację czy dane są podpięte do systemu
*)
METHOD PUBLIC IsInit : BOOL
VAR_INPUT
END_VAR
IsInit			:= THIS^.bIsInit;
END_METHOD

METHOD PUBLIC IsLinkedReferences : BOOL
VAR_INPUT
END_VAR
IF (__ISVALIDREF (THIS^.refstBaseLoggerElementDataHMI)) THEN
	IsLinkedReferences			:= TRUE;
END_IF
END_METHOD

(*			
	RAFALOS
	Rafał Osajda		23.09.2025		TC 4024.66
	Zwraca flagę przypisywaną w FB_Init tworzonego elementu
*)
METHOD IsValidData : BOOL
VAR_INPUT
END_VAR
IsValidData				:= THIS^.bIsValidData;
END_METHOD

(*			
	RafalOS
	Rafał Osajda		14.11.2025		TC 4024.66
	Metoda przygotowywania danych dla HMI 
	W niej odbywa się odpytywanie właściego elementu przez łącznik
*)
METHOD PUBLIC PrepareDataForHMI : BOOL
VAR_INPUT
END_VAR
END_METHOD

(*			
	RafalOS
	Rafał Osajda		19.11.2025		TC 4024.66
	Przygotowanie ramki pood tamke do wyświetlenia - tylko przygotowanie a nie przygotowanie danych do wyświetlenia
*)
METHOD PUBLIC PrepareForScreen : BOOL
VAR_INPUT
END_VAR
END_METHOD

METHOD PRIVATE PrepareQuantitiesForDisplay : BOOL
VAR_INPUT
	stCounted			: ST_BaseEvents_ActiveEvents;
	stFromLogger		: ST_BaseEvents_ActiveEvents;
END_VAR

VAR
	iI: INT;
	stmp1: STRING;
END_VAR
stmp1	:= CONCAT (stmp1,TO_STRING (stCounted.iNumberOfActiveWithConfirmation));
stmp1	:= CONCAT (stmp1, '/');
stmp1	:= CONCAT (stmp1, TO_STRING (stFromLogger.iNumberOfActiveWithConfirmation));

THIS^.refstBaseLoggerElementDataHMI.stButtons.sAcknowledgeAll		:= stmp1;
THIS^.refstBaseLoggerElementDataHMI.stButtons.sAcknowledgeSelected	:= '1/1';

stmp1	:= CONCAT ('',TO_STRING (stCounted.iNumberOfActive));
stmp1	:= CONCAT (stmp1, '/');
stmp1	:= CONCAT (stmp1, TO_STRING (stFromLogger.iNumberOfActive));
THIS^.refstBaseLoggerElementDataHMI.stButtons.sCloseAll				:= stmp1;
THIS^.refstBaseLoggerElementDataHMI.stButtons.sCloseSelected		:= '1/1';

FOR iI := 1	TO GVL_BaseConstans.NUMBER_OF_EVENT_CATEGORIES DO
	THIS^.refstBaseLoggerElementDataHMI.stFilter.arrTextOnEventCategory [iI]	:= 
		CONCAT (TO_STRING (stCounted.arrTotalNumer [iI]), CONCAT ('/',TO_STRING (stFromLogger.arrTotalNumer [iI])));
END_FOR
END_METHOD

METHOD PRIVATE RemoveRowFormList : BOOL
VAR_INPUT
	refstFilter				: REFERENCE TO ST_BaseHMIConnectorEvents_Filter;
	uiIDEvent				: UINT;
	uiIDItem				: UINT;
	bActive					: BOOL;
	stItemInformation		: ST_BaseLogger_ItemDataToDisplay;
END_VAR
VAR
	bRemove					: BOOL;
	iK						: INT;
	bRemoveHelp				: BOOL;
END_VAR
bRemove		:= FALSE;
bRemove		:= bRemove OR (refstFilter.bActive AND NOT bActive);
bRemove		:= bRemove OR (refstFilter.bNotActive AND bActive);
bRemove		:= bRemove OR (refstFilter.bIDItem	AND uiIDItem <> refstFilter.uiIDItem);
bRemove		:= bRemove OR (refstFilter.bIDEvent AND 
uiIDEvent <> refstFilter.uiIDEvent);
FOR iK := 1 TO GVL_BaseConstans.NUMBER_OF_EVENT_CATEGORIES DO
	CASE iK OF 
		E_BaseEvents_Category.Error		: bRemoveHelp	:=  stItemInformation.eEventCategory = E_BaseEvents_Category.Error;
		E_BaseEvents_Category.Alarm		: bRemoveHelp	:=  stItemInformation.eEventCategory = E_BaseEvents_Category.Alarm;
		E_BaseEvents_Category.Safety	: bRemoveHelp	:=  stItemInformation.eEventCategory = E_BaseEvents_Category.Safety;
		E_BaseEvents_Category.Message	: bRemoveHelp	:=  stItemInformation.eEventCategory = E_BaseEvents_Category.Message;
	END_CASE
	bRemove		:= bRemove OR (refstFilter.arrSelectedEventCategory [iK] AND bRemoveHelp);
END_FOR
//przeddział czasowy

RemoveRowFormList	:= bRemove;
END_METHOD

METHOD PROTECTED SelectLocation : WSTRING
VAR_INPUT
	stTexts			: ST_BaseLabel;
	eLocation		: E_BaseLocation;
END_VAR
SelectLocation := stTexts.arrText [eLocation];
END_METHOD

END_FUNCTION_BLOCK

// ---- POUs/A03b_FB_BaseHMILoggerElement_Command/FB_BaseHMILoggerElement_Command.TcPOU
FUNCTION_BLOCK FB_BaseHMILoggerElement_Command
VAR
	stDataCheck					: ST_BaseHMILoggerElement_Command_DataCheck;

END_VAR

END_FUNCTION_BLOCK

// ---- POUs/A04a_FB_BaseHMIComponent_View/FB_BaseHMIComponent_View.TcPOU
FUNCTION_BLOCK FB_BaseHMIComponent_View EXTENDS FB_BaseHMILoggerElement_View IMPLEMENTS ITF_BaseHMIComponent_View
VAR
	itfBaseComponentConnector			: ITF_BaseComponent_HMI_Connector;
	refstBaseComponentDataHMI			: REFERENCE TO ST_BaseHMIComponent_View;
END_VAR

METHOD PUBLIC IsLinkedReferences : BOOL
VAR_INPUT
END_VAR
IF (SUPER^.IsLinkedReferences () AND __ISVALIDREF (THIS^.refstBaseComponentDataHMI)) THEN
	IsLinkedReferences			:= TRUE;
END_IF
END_METHOD

METHOD PUBLIC JoinTheList : INT
VAR_INPUT
	refstList				: REFERENCE TO ST_ListOfElement_HMI;
	iNumberOfParent			: INT; 	//numer rodzica na liście
END_VAR
IF (refstList.iNumberOfAdded + 1 <= TO_INT (GVL_BaseConstans.MAX_NUMBER_OF_ALL_ITEM) AND THIS^.itfBaseComponentConnector <> 0) THEN
	refstList.iNumberOfAdded := refstList.iNumberOfAdded + 1;
	refstList.arrRow [refstList.iNumberOfAdded].stIdentifiers := THIS^.itfBaseComponentConnector.GetIdentyfier ();
	refstList.arrRow [refstList.iNumberOfAdded].itfElement := THIS^;
	IF (refstList.arrRow [refstList.iNumberOfAdded].stIdentifiers.eType = E_BaseElementType.eTop) THEN
		(*	Zapisujemy w tablicy arrListaPB indekxy PB	*)
		refstList.iNumberOfAddedTE := refstList.iNumberOfAddedTE + 1;
		refstList.arrRowOfListTE [refstList.iNumberOfAddedTE] := refstList.iNumberOfAdded;
		JoinTheList := refstList.iNumberOfAdded;
	ELSE
		(*	Dopisanie numeru swojego indeksu do poprzedniego idneksu czyli do swojego rodzica 	*)
		refstList.arrRow [iNumberOfParent].iNumberOfChildAdded := refstList.arrRow [iNumberOfParent].iNumberOfChildAdded + 1;
		refstList.arrRow [iNumberOfParent].arrChild [refstList.arrRow [iNumberOfParent].iNumberOfChildAdded] := refstList.iNumberOfAdded;
		JoinTheList := refstList.iNumberOfAdded;
	END_IF
END_IF
END_METHOD

(*			
	RafalOS
	Rafał Osajda		14.11.2025		TC 4024.66
	Metoda przygotowywania danych dla HMI 
	W niej odbywa się odpytywanie właściego elementu przez łącznik
*)
METHOD PUBLIC PrepareDataForHMI : BOOL
VAR_INPUT
END_VAR
THIS^.refstBaseComponentDataHMI.wsName := THIS^.GetTextFromLabelForActiveLocation (stLabel := THIS^.itfBaseComponentConnector.GetName ());
END_METHOD

END_FUNCTION_BLOCK

// ---- POUs/A04b_FB_BaseHMIComponent_Command/FB_BaseHMIComponent_Command.TcPOU
(*			
	RafalOS
	Rafał Osajda		19.12.2025		TC 4024.66
	Obsługa sterowania z HMI testowanie czy można uzyć rozkazu i przekazać do dalej do elementu logicznego
*)
FUNCTION_BLOCK FB_BaseHMIComponent_Command EXTENDS FB_BaseHMILoggerElement_Command IMPLEMENTS ITF_BaseHMIComponent_Command
VAR
//	itfParent					: itf_basecontrolelement_command_; w komponencie musi byc itf do rodzica by się spytac czy można się ruszać czy coś innego się nei rusza 
	
END_VAR

END_FUNCTION_BLOCK

// ---- POUs/A05a_FB_BaseHMIControlElement_View/FB_BaseHMIControlElement_View.TcPOU
FUNCTION_BLOCK FB_BaseHMIControlElement_View EXTENDS FB_BaseHMIComponent_View IMPLEMENTS ITF_BaseHMIControlElement_View
VAR
	itfBaseControlElementConnector		: ITF_BaseControlElement_HMI_Connector;
	refstBaseControlElementDataHMI		: REFERENCE TO ST_BaseHMIControlElement_View;
	(*	lista componentów składających się na ten element w elemencie docelowym dodać itf dla konkretnych elementów	*)
	arrComponent						: ARRAY  [1..GVL_BaseConstans.MAX_ITEM_PER_ELEMENT] OF ITF_BaseHMIComponent_View;
	uiNumberOfComponents				: UINT;

END_VAR

METHOD PROTECTED AddComponent : BOOL
VAR_INPUT
	itfComponentHMI				: ITF_BaseHMIComponent_View;
END_VAR
IF (THIS^.uiNumberOfComponents + 1 <= GVL_BaseConstans.MAX_ITEM_PER_ELEMENT) THEN
	THIS^.uiNumberOfComponents		:= THIS^.uiNumberOfComponents + 1;
	THIS^.arrComponent [THIS^.uiNumberOfComponents]	:= itfComponentHMI;
	AddComponent				:= TRUE;
ELSE
	;//zwrocenie zbyt dużo komponentow
END_IF
END_METHOD

METHOD PUBLIC IsLinkedReferences : BOOL
VAR_INPUT
END_VAR
IF (SUPER^.IsLinkedReferences () AND __ISVALIDREF (THIS^.refstBaseControlElementDataHMI)) THEN
	IsLinkedReferences			:= TRUE;
END_IF
END_METHOD

METHOD PUBLIC IsValidCommonData : BOOL
VAR_INPUT
END_VAR

VAR
	bResult: BOOL;
	iI: INT;
END_VAR
bResult						:= SUPER^.IsValidCommonData ();

FOR iI := 1 TO TO_INT (THIS^.uiNumberOfComponents) DO
	bResult					:= bResult AND THIS^.arrComponent [iI].IsValidCommonData ();
END_FOR

IsValidCommonData			:= bResult;
END_METHOD

METHOD PUBLIC JoinTheList : INT
VAR_INPUT
	refstList				: REFERENCE TO ST_ListOfElement_HMI;
	iNumberOfParent			: INT; 	//numer rodzica na liście
END_VAR
VAR
	iI						: INT;
	itmpNumberOfParent		: INT;
END_VAR
itmpNumberOfParent	:= SUPER^.JoinTheList (refstList := refstList, iNumberOfParent := iNumberOfParent);

FOR iI := 1 TO TO_INT (THIS^.uiNumberOfComponents) DO
	THIS^.arrComponent [iI].JoinTheList (refstList := refstList, iNumberOfParent := itmpNumberOfParent);
END_FOR

JoinTheList	:= itmpNumberOfParent;
END_METHOD

METHOD PUBLIC LinkCommonData : BOOL
VAR_INPUT
	stCommonData				: REFERENCE TO ST_BaseCommonData;
END_VAR
VAR
	bResult						: BOOL;
	iI: INT;
END_VAR
bResult							:= SUPER^.LinkCommonData (stCommonData := stCommonData);

FOR iI := 1 TO TO_INT (THIS^.uiNumberOfComponents) DO
	bResult := bResult AND THIS^.arrComponent [iI].LinkCommonData (stCommonData := stCommonData);
END_FOR

LinkCommonData					:= bResult;
END_METHOD

END_FUNCTION_BLOCK

// ---- POUs/A05b_FB_BaseHMIControlElement_Command/FB_BaseHMIControlElement_Command.TcPOU
FUNCTION_BLOCK FB_BaseHMIControlElement_Command EXTENDS FB_BaseHMIComponent_Command IMPLEMENTS ITF_BaseHMIControlElement_Command
VAR
END_VAR

END_FUNCTION_BLOCK

// ---- POUs/A06a_FB_BaseHMIGroupElement_View/FB_BaseHMIGroupElement_View.TcPOU
FUNCTION_BLOCK FB_BaseHMIGroupElement_View EXTENDS FB_BaseHMIControlElement_View IMPLEMENTS ITF_BaseHMIGroupElement_View
VAR
	itfBaseGroupElementConnector		: ITF_BaseGroupElement_HMI_Connector;
	refstBaseGroupElementDataHMI		: REFERENCE TO ST_BaseHMIGroupElement_View;
	(*	lista elementów składających się na ten element w elemencie docelowym dodać itf dla konkretnych elementów	*)
	arrControlElement					: ARRAY [1..GVL_BaseConstans.MAX_ITEM_PER_ELEMENT] OF ITF_BaseHMIControlElement_View;
	uiNumberOfControlElement			: UINT;
END_VAR

METHOD PROTECTED AddControlElement : BOOL
VAR_INPUT
	itfControlElementHMI		: ITF_BaseHMIControlElement_View;
END_VAR
IF (THIS^.uiNumberOfControlElement + 1 <= GVL_BaseConstans.MAX_ITEM_PER_ELEMENT) THEN
	THIS^.uiNumberOfControlElement		:= THIS^.uiNumberOfControlElement + 1;
	THIS^.arrControlElement [THIS^.uiNumberOfControlElement]	:= itfControlElementHMI;
	AddControlElement			:= TRUE;
ELSE
	;//zwrocenie zbyt dużo komponentow
END_IF
END_METHOD

METHOD PUBLIC IsLinkedReferences : BOOL
VAR_INPUT
END_VAR
IF (SUPER^.IsLinkedReferences () AND __ISVALIDREF (THIS^.refstBaseGroupElementDataHMI)) THEN
	IsLinkedReferences			:= TRUE;
END_IF
END_METHOD

METHOD PUBLIC IsValidCommonData : BOOL
VAR_INPUT
END_VAR

VAR
	bResult: BOOL;
	iI: INT;
END_VAR
bResult						:= SUPER^.IsValidCommonData ();

FOR iI := 1 TO TO_INT (THIS^.uiNumberOfControlElement) DO
	bResult					:= bResult AND THIS^.arrControlElement [iI].IsValidCommonData ();
END_FOR

IsValidCommonData			:= bResult;
END_METHOD

METHOD PUBLIC JoinTheList : INT
VAR_INPUT
	refstList				: REFERENCE TO ST_ListOfElement_HMI;
	iNumberOfParent			: INT; 	//numer rodzica na liście
END_VAR
VAR
	iI						: INT;
	itmpNumberOfParent			: INT;
END_VAR
itmpNumberOfParent		:= SUPER^.JoinTheList (refstList := refstList, iNumberOfParent := iNumberOfParent);

FOR iI := 1 TO TO_INT (THIS^.uiNumberOfControlElement) DO
	THIS^.arrControlElement [iI].JoinTheList (refstList := refstList, iNumberOfParent := itmpNumberOfParent);
END_FOR

JoinTheList	:= itmpNumberOfParent;
END_METHOD

METHOD PUBLIC LinkCommonData : BOOL
VAR_INPUT
	stCommonData				: REFERENCE TO ST_BaseCommonData;
END_VAR
VAR
	bResult						: BOOL;
	iI: INT;
END_VAR
bResult							:= SUPER^.LinkCommonData (stCommonData := stCommonData);

FOR iI := 1 TO TO_INT (THIS^.uiNumberOfControlElement) DO
	bResult := bResult AND THIS^.arrControlElement [iI].LinkCommonData (stCommonData := stCommonData);
END_FOR

LinkCommonData					:= bResult;
END_METHOD

END_FUNCTION_BLOCK

// ---- POUs/A06b_FB_BaseHMIGroupElement_Command/FB_BaseHMIGroupElement_Command.TcPOU
FUNCTION_BLOCK FB_BaseHMIGroupElement_Command EXTENDS FB_BaseHMIControlElement_Command IMPLEMENTS ITF_BaseHMIGroupElement_Command
VAR
END_VAR

END_FUNCTION_BLOCK

// ---- POUs/A07a_FB_BaseHMITopElement_View/FB_BaseHMITopElement_View.TcPOU
FUNCTION_BLOCK FB_BaseHMITopElement_View EXTENDS FB_BaseHMIGroupElement_View IMPLEMENTS ITF_BaseHMITopElement_View
VAR
	itfBaseTopElementConnector			: ITF_BaseTopElement_HMI_Connector;
	refstBaseTopElementDataHMI			: REFERENCE TO ST_BaseHMITopElement_View;
END_VAR

METHOD PUBLIC IsLinkedReferences : BOOL
VAR_INPUT
END_VAR
IF (SUPER^.IsLinkedReferences () AND __ISVALIDREF (THIS^.refstBaseTopElementDataHMI)) THEN
	IsLinkedReferences			:= TRUE;
END_IF
END_METHOD

END_FUNCTION_BLOCK

// ---- POUs/A07b_FB_BaseHMITopElement_Command/FB_BaseHMITopElement_Command.TcPOU
FUNCTION_BLOCK FB_BaseHMITopElement_Command EXTENDS FB_BaseHMIGroupElement_Command IMPLEMENTS ITF_BaseHMITopElement_Command
VAR
END_VAR

END_FUNCTION_BLOCK

// ---- POUs/B02_Recipe/FB_BaseRecipe_HMI.TcPOU
FUNCTION_BLOCK FB_BaseRecipe_HMI EXTENDS FB_Base IMPLEMENTS ITF_BaseRecipe_HMI
VAR
	itfBaseRecipe			: ITF_BaseRecipe_HMI_Connector;
	refstRepiceData			: REFERENCE TO ST_BaseRecipe_HMI;
	
END_VAR

(*			
	RafalOS
	Rafał Osajda		03.03.2025		TC 4026.13		wer. 0.0.0.1
	Kopiuje składniki z wybranej receptury i tworzy nową recepture
*)
METHOD PUBLIC AddRecipeFromRecipe : BOOL
VAR_INPUT
	uiNumberRecipe				: UINT;
	stTexts						: ST_BaseLabel;
END_VAR
THIS^.itfBaseRecipe.AddRecipeFromRecipe (
	uiNumberRecipe 	:= uiNumberRecipe,
	stTexts			:= stTexts
);
END_METHOD

(*			
	RafalOS
	Rafał Osajda		03.03.2025		TC 4026.13		wer. 0.0.0.1
	Kopiuje składniki z wybranego szablonu i tworzy nową recepture
*)
METHOD PUBLIC AddRecipeFromTemplate : BOOL
VAR_INPUT
	uiNumberTemplates			: UINT;
	stTexts						: ST_BaseLabel;
END_VAR
THIS^.itfBaseRecipe.AddRecipeFromTemplate (
	uiNumberTemplates 	:= uiNumberTemplates,
	stTexts				:= stTexts
);
END_METHOD

(*			
	RafalOS
	Rafał Osajda		03.06.2025		TC 4024.66
	usuwa referencje do wybranej
*)
METHOD PUBLIC ClearChosen
VAR_INPUT
END_VAR
THIS^.itfBaseRecipe.ClearChosen ();
END_METHOD

(*			
	RafalOS
	Rafał Osajda		25.10.2025		TC 4024.66
	Utworzenie nowych szablonów receptur na podstawie dodanych fb zewnętrznych - wywołanie metody powoduje
	skosowanie dotychczasowych szablonów i receptur
*)
METHOD PUBLIC CreateRecipeTemplates : BOOL
VAR_INPUT
END_VAR
THIS^.itfBaseRecipe.CreateTemplates ();
END_METHOD

(*			
	RafalOS
	Rafał Osajda		03.03.2025		TC 4026.13		wer. 0.0.0.1
	
*)
METHOD PUBLIC DeleteRecipe : BOOL
VAR_INPUT
	uiNumber				: uint;
END_VAR
THIS^.itfBaseRecipe.DeleteRecipe (uiNumber := uiNumber);
END_METHOD

METHOD FB_init : BOOL
VAR_INPUT
	bInitRetains : BOOL; // if TRUE, the retain variables are initialized (warm start / cold start)
	bInCopyCode : BOOL;  // if TRUE, the instance afterwards gets moved into the copy code (online change)
	fbBaseRecipe			: ITF_BaseRecipe_HMI_Connector;
END_VAR
THIS^.itfBaseRecipe := fbBaseRecipe;
END_METHOD

(*			
	RafalOS
	Rafał Osajda		03.03.2025		TC 4026.13		wer. 0.0.0.1
	
*)
METHOD PUBLIC GetIngredientFromRecipe : ST_BaseDescriptor
VAR_INPUT
	uiNumberOfRecipe			: UINT;
	uiNumberOfIngredient		: UINT;
END_VAR
GetIngredientFromRecipe			:= THIS^.itfBaseRecipe.GetIngredientFromRecipe (
									uiNumberOfRecipe := uiNumberOfRecipe,
									uiNumberOfIngredient := uiNumberOfIngredient
								);
END_METHOD

(*			
	RafalOS
	Rafał Osajda		02.12.2025		TC 4024.66
	Zwraca do tablicy wybrany zakres składników
*)
METHOD PUBLIC GetIngredientRange 
VAR_INPUT
	iRecipe			: INT;	//numer receptury z której bierzemy składniki
	iStartIndex		: INT;	//numer startowy składnika
	iCount			: INT;	//ilośc pobieranych 
END_VAR
VAR_IN_OUT
	arrOut : ARRAY [*] OF ST_BaseDescriptor;
END_VAR
VAR_OUTPUT
	iNumberOfFilledData	: INT;	//ilosc wypelnionych danych na strone
END_VAR
THIS^.itfBaseRecipe.GetIngredientRange (
	iRecipe		:= iRecipe,
	iStartIndex	:= iStartIndex,
	iCount		:= iCount,
	arrOut		:= arrOut,
	iNumberOfFilledData	=> iNumberOfFilledData
);
END_METHOD

METHOD GetNameList : ST_BaseRecipeList
VAR_INPUT
END_VAR
GetNameList := THIS^.itfBaseRecipe.GetNameList ();
END_METHOD

METHOD GetNameListTemplate : ST_BaseRecipeList
VAR_INPUT
END_VAR
GetNameListTemplate := THIS^.itfBaseRecipe.GetNameListTemplate ();
END_METHOD

METHOD GetNamesOfSelectRecipe : ST_BaseLabel
VAR_INPUT

END_VAR
GetNamesOfSelectRecipe := THIS^.itfBaseRecipe.GetNamesOfSelectRecipe ();
END_METHOD

(*			
	RafalOS
	Rafał Osajda		03.03.2025		TC 4026.13		wer. 0.0.0.1
	
*)
METHOD PUBLIC GetNumberIngredientOfRecipe : UINT
VAR_INPUT
	uiNumber				: UINT;
END_VAR
GetNumberIngredientOfRecipe 		:= THIS^.itfBaseRecipe.GetNumberIngredientOfRecipe (uiNumber := uiNumber);
END_METHOD

METHOD PUBLIC GetNumberOfChoosen : UINT
VAR_INPUT
END_VAR
GetNumberOfChoosen := THIS^.itfBaseRecipe.GetNumberOfChoosen ();
END_METHOD

METHOD PUBLIC GetNumberOfRecipe : UINT
VAR_INPUT
END_VAR
GetNumberOfRecipe			:= THIS^.itfBaseRecipe.GetNumberOfRecipe ();
END_METHOD

METHOD PUBLIC GetNumberOfTemplate : UINT
VAR_INPUT
END_VAR
GetNumberOfTemplate		:= THIS^.itfBaseRecipe.GetNumberOfTemplate ();
END_METHOD

(*			
	RafalOS
	Rafał Osajda		06.12.2025		TC 4024.66
	Sprawdza czy receptrua została wybrana
*)
METHOD PUBLIC IsRecipeSelected : BOOL
VAR_INPUT
END_VAR
IsRecipeSelected := THIS^.itfBaseRecipe.IsChoosen ();
END_METHOD

METHOD PUBLIC LinkRecipeDataHMI : BOOL
VAR_INPUT
	stRecipe			: REFERENCE TO ST_BaseRecipe_HMI;
END_VAR
THIS^.refstRepiceData REF= stRecipe;
END_METHOD

(*			
	RafalOS
	Rafał Osajda		06.12.2025		TC 4024.66
	Wybranie receputury
*)
METHOD SelectRecipe : BOOL
VAR_INPUT
	uiRecipe: UINT;
END_VAR
THIS^.itfBaseRecipe.Choose (
	uiNumber := uiRecipe
);
END_METHOD

(*			
	RafalOS
	Rafał Osajda		05.12.2025		TC 4024.66
	Ustawia nową wartośc w podanym składniku
*)
METHOD PUBLIC SetIngredientValue
VAR_INPUT
	iRecipe			: int;
	iIngredient		: INT;
	rValue			: REAL;
END_VAR
THIS^.itfBaseRecipe.SetIngredientValue (
	iRecipe := iRecipe,
	iIngredient := iIngredient,
	rValue := rValue
);
END_METHOD

END_FUNCTION_BLOCK
